// TIA Portal V19 export
DATA_BLOCK "DEBUG_MES_Receive_Msg_Topic3XX"   // DB203
// stored: MemoryReserve 100
   VAR
      DEBUG_RECEIVE { ExternalAccessible := 'False'; ExternalVisible := 'False'; ExternalWritable := 'False'} : Struct
         Enable : Bool;
         AckChangeStep : Bool;
         ActualStep : Int;
      END_STRUCT;
      ACK_MSG_enable : Bool;
      NEW_MSG_300 : Struct
         ABILITA_FC : Bool;
         EXE_MSG : Bool;
         MSG : "MES_Msg";
      END_STRUCT;
      NEW_MSG_301 : Struct
         ABILITA_FC : Bool;
         EXE_MSG : Bool;
         MSG : "MES_Msg";
      END_STRUCT;
   END_VAR
BEGIN
END_DATA_BLOCK
